Fanuc KAREL source: kt00057.KL

-- PROVISIONAL review KL for V1013-1; original PC SHA256 c628ac5144c1fa4790afe9f2bbdaefc3ccdc01f5931e1033e580e0bd4fa49025
-- Incomplete behavior may be omitted. Consult companion uncertainty JSON. Do not deploy.
PROGRAM KT00057
%NOLOCKGROUP
VAR
  I2 : INTEGER
  OUT : INTEGER
-- UNRESOLVED_DECL H1 type=002017
BEGIN
  -- UNRESOLVED_PC offsets 5-19; opcodes 2E,22,9D,33,B4
  -- UNRESOLVED_PC offsets 24-35; opcodes 2E,23
  -- UNRESOLVED_PC offsets 40-62; opcodes 22,9D,33,B3,21,53,23
  -- UNRESOLVED_PC offsets 67-71; opcodes 7F
END KT00057
